(* PLC project KEVIN, Unknown Unnamed 1 *)
(* stored: creationDateTime 2021-12-14T14:39:40, modificationDateTime 2022-01-31T14:09:18 *)

PROGRAM DualCarElevator
  VAR
    C1F1LimitSw AT %IX0.0 : BOOL;
    C2F1LimitSw AT %IX0.1 : BOOL;
    C2F2LimitSw AT %IX0.3 : BOOL;
    C2F3LimitSw AT %IX0.5 : BOOL;
    C2F4LimitSw AT %IX0.7 : BOOL;
    F2DownCall AT %QX0.5 : BOOL;
  END_VAR
  VAR
    C2F1MemLoc : BOOL;
    C2F2MemLoc : BOOL;
    C2F3MemLoc : BOOL;
    C2F4MemLoc : BOOL;
    C2F1VisMem : BOOL;
    C2F2VisMem : BOOL;
    C2F3VisMem : BOOL;
    C2F4VisMem : BOOL;
    C2F1LastVisMem : BOOL;
    C2F2LastVisMem : BOOL;
    C2F3LastVisMem : BOOL;
    C2F4LastVisMem : BOOL;
  END_VAR
  VAR
    C2MotorUp AT %QX0.2 : BOOL;
    C2MotorDown AT %QX0.3 : BOOL;
  END_VAR
  VAR
    C2MotorStops : BOOL;
    C2DoorOpenReady : BOOL;
    C2DoorClose : BOOL;
    C2DoorOpen : BOOL;
    C2DoorIsClosed : BOOL;
    C2DoorCloseReady : BOOL;
  END_VAR
  VAR
    C2F1CarCall AT %QX100.4 : BOOL;
    C2F2CarCall AT %QX100.5 : BOOL;
    C2F3CarCall AT %QX100.6 : BOOL;
    C2F4CarCall AT %QX100.7 : BOOL;
    F2UpCall AT %QX0.6 : BOOL;
    F3UpCall AT %QX1.0 : BOOL;
    F3DownCall AT %QX0.7 : BOOL;
    C1F2LimitSw AT %IX0.2 : BOOL;
    C1F3LimitSw AT %IX0.4 : BOOL;
    C1F4LimitSw AT %IX0.6 : BOOL;
    C1F1CarCall AT %QX100.0 : BOOL;
    C1F2CarCall AT %QX100.1 : BOOL;
    C1F3CarCall AT %QX100.2 : BOOL;
    C1F4CarCall AT %QX100.3 : BOOL;
    F1UpCall AT %QX0.4 : BOOL;
    F4DownCall AT %QX1.1 : BOOL;
    C1MotorUp AT %QX0.0 : BOOL;
    C1MotorDown AT %QX0.1 : BOOL;
  END_VAR
  VAR
    C1MotorStops : BOOL;
    C1DoorOpen : BOOL;
    C1DoorClose : BOOL;
    C1F1MemLoc : BOOL;
    C1F2MemLoc : BOOL;
    C1F3MemLoc : BOOL;
    C1F4MemLoc : BOOL;
    C1F1LastVisMem : BOOL;
    C1F2LastVisMem : BOOL;
    C1F3LastVisMem : BOOL;
    C1F4LastVisMem : BOOL;
    C1F1VisMem : BOOL;
    C1F2VisMem : BOOL;
    C1F3VisMem : BOOL;
    C1F4VisMem : BOOL;
    DoorOpenDelay : TON;
    C1DoorOpenReady : BOOL;
    C1DoorCloseReady : BOOL;
    C1DoorIsClosed : BOOL;
    C1DoorOpeningDelay : TON;
    C1DoorClosingDelay : TON;
    DoorOpenDelay0 : TON;
    C2DoorClosingDelay : TON;
    C2DoorOpeningDelay : TON;
  END_VAR
  VAR
    C1F1CarBtn AT %IX100.0 : BOOL;
    C1F2CarBtn AT %IX100.1 : BOOL;
    C1F3CarBtn AT %IX100.2 : BOOL;
    C1F4CarBtn AT %IX100.3 : BOOL;
    C2F1CarBtn AT %IX100.5 : BOOL;
    C2F2CarBtn AT %IX100.6 : BOOL;
    C2F3CarBtn AT %IX100.7 : BOOL;
    C2F4CarBtn AT %IX101.0 : BOOL;
    F1UpBtn AT %IX1.0 : BOOL;
    F2DownBtn AT %IX1.1 : BOOL;
    F2UpBtn AT %IX1.2 : BOOL;
    F3DownBtn AT %IX1.3 : BOOL;
    F3UpBtn AT %IX1.4 : BOOL;
    F4DownBtn AT %IX1.5 : BOOL;
  END_VAR
  VAR  (* added by the conversion: wires and edge detectors of the diagram *)
    F_TRIG1 : F_TRIG;
    F_TRIG2 : F_TRIG;
    F_TRIG3 : F_TRIG;
    F_TRIG4 : F_TRIG;
    F_TRIG5 : F_TRIG;
    F_TRIG6 : F_TRIG;
    F_TRIG7 : F_TRIG;
    F_TRIG8 : F_TRIG;
  END_VAR

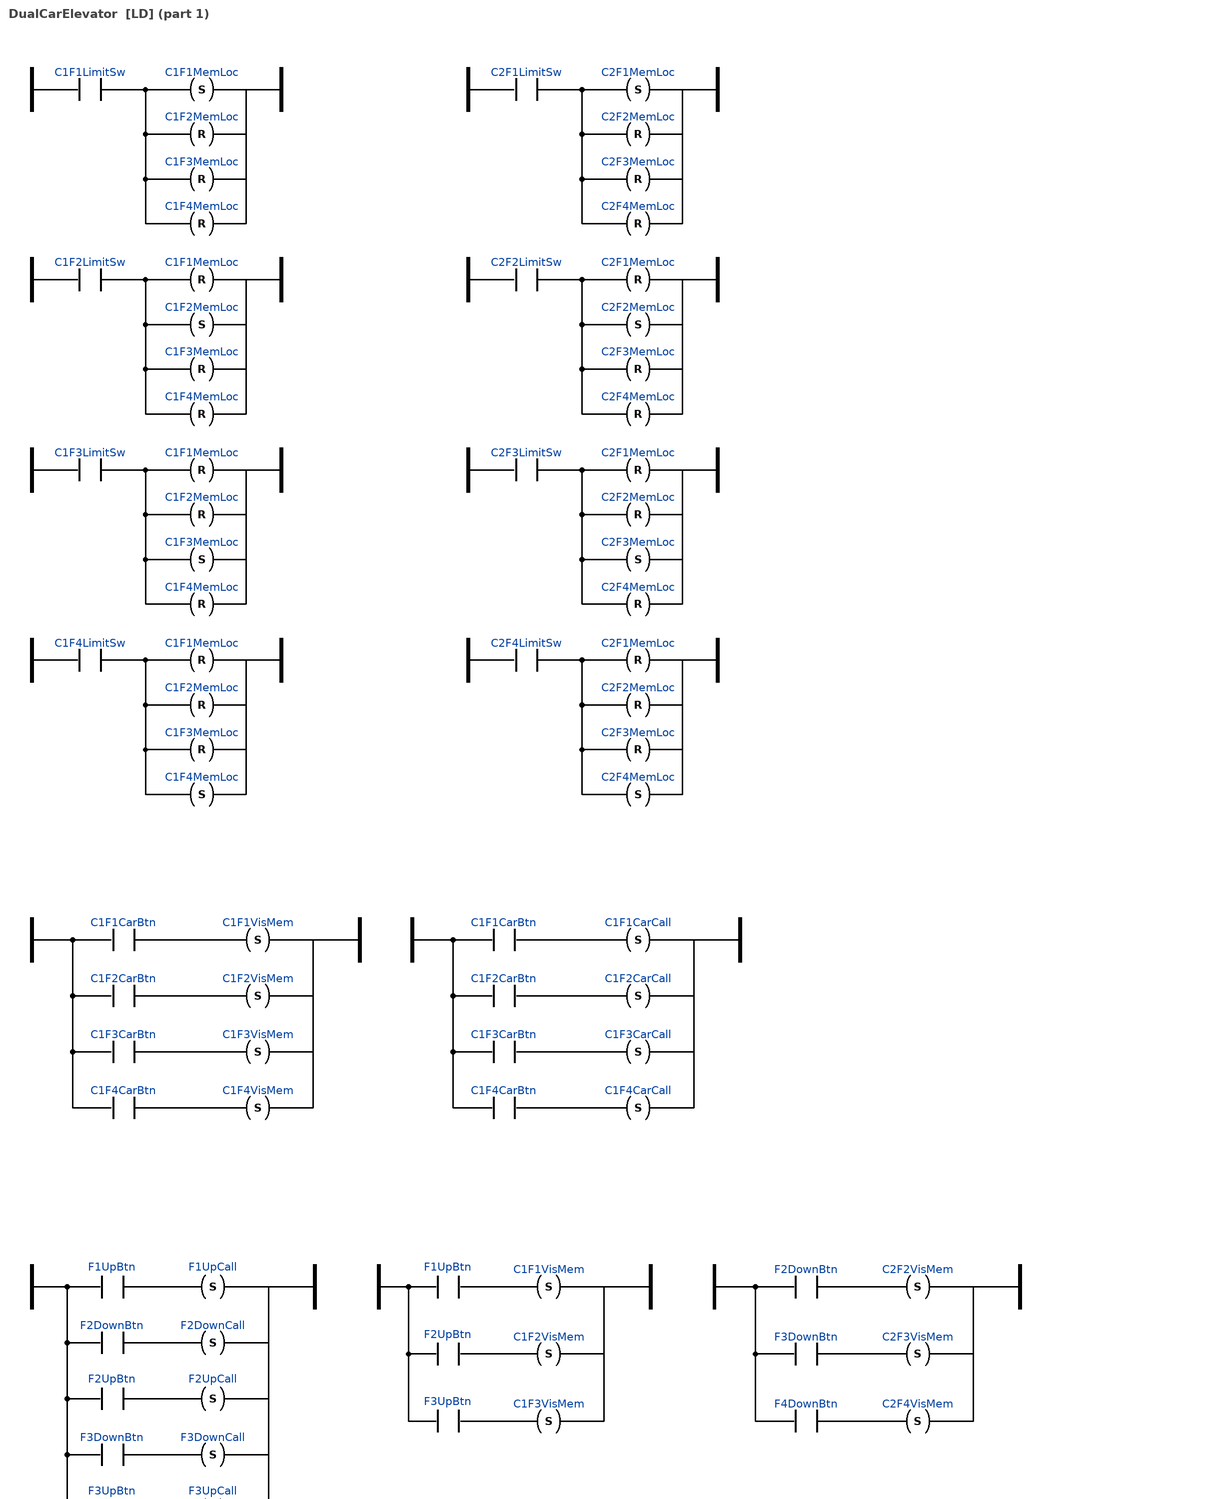
(* LD diagram, written out as Structured Text *)
IF C1F1LimitSw THEN C1F1MemLoc := TRUE; END_IF;
IF C2F1LimitSw THEN C2F1MemLoc := TRUE; END_IF;
IF C1F1LimitSw THEN C1F2MemLoc := FALSE; END_IF;
IF C2F1LimitSw THEN C2F2MemLoc := FALSE; END_IF;
IF C1F1LimitSw THEN C1F3MemLoc := FALSE; END_IF;
IF C2F1LimitSw THEN C2F3MemLoc := FALSE; END_IF;
IF C1F1LimitSw THEN C1F4MemLoc := FALSE; END_IF;
IF C2F1LimitSw THEN C2F4MemLoc := FALSE; END_IF;
IF C1F2LimitSw THEN C1F1MemLoc := FALSE; END_IF;
IF C2F2LimitSw THEN C2F1MemLoc := FALSE; END_IF;
IF C1F2LimitSw THEN C1F2MemLoc := TRUE; END_IF;
IF C2F2LimitSw THEN C2F2MemLoc := TRUE; END_IF;
IF C1F2LimitSw THEN C1F3MemLoc := FALSE; END_IF;
IF C2F2LimitSw THEN C2F3MemLoc := FALSE; END_IF;
IF C1F2LimitSw THEN C1F4MemLoc := FALSE; END_IF;
IF C2F2LimitSw THEN C2F4MemLoc := FALSE; END_IF;
IF C1F3LimitSw THEN C1F1MemLoc := FALSE; END_IF;
IF C2F3LimitSw THEN C2F1MemLoc := FALSE; END_IF;
IF C1F3LimitSw THEN C1F2MemLoc := FALSE; END_IF;
IF C2F3LimitSw THEN C2F2MemLoc := FALSE; END_IF;
IF C1F3LimitSw THEN C1F3MemLoc := TRUE; END_IF;
IF C2F3LimitSw THEN C2F3MemLoc := TRUE; END_IF;
IF C1F3LimitSw THEN C1F4MemLoc := FALSE; END_IF;
IF C2F3LimitSw THEN C2F4MemLoc := FALSE; END_IF;
IF C1F4LimitSw THEN C1F1MemLoc := FALSE; END_IF;
IF C2F4LimitSw THEN C2F1MemLoc := FALSE; END_IF;
IF C1F4LimitSw THEN C1F2MemLoc := FALSE; END_IF;
IF C2F4LimitSw THEN C2F2MemLoc := FALSE; END_IF;
IF C1F4LimitSw THEN C1F3MemLoc := FALSE; END_IF;
IF C2F4LimitSw THEN C2F3MemLoc := FALSE; END_IF;
IF C1F4LimitSw THEN C1F4MemLoc := TRUE; END_IF;
IF C2F4LimitSw THEN C2F4MemLoc := TRUE; END_IF;
IF C1F1CarBtn THEN C1F1VisMem := TRUE; END_IF;
IF C1F1CarBtn THEN C1F1CarCall := TRUE; END_IF;
IF C1F2CarBtn THEN C1F2VisMem := TRUE; END_IF;
IF C1F2CarBtn THEN C1F2CarCall := TRUE; END_IF;
IF C1F3CarBtn THEN C1F3VisMem := TRUE; END_IF;
IF C1F3CarBtn THEN C1F3CarCall := TRUE; END_IF;
IF C1F4CarBtn THEN C1F4VisMem := TRUE; END_IF;
IF C1F4CarBtn THEN C1F4CarCall := TRUE; END_IF;
IF F1UpBtn THEN F1UpCall := TRUE; END_IF;
IF F1UpBtn THEN C1F1VisMem := TRUE; END_IF;
IF F2DownBtn THEN C2F2VisMem := TRUE; END_IF;
IF F2DownBtn THEN F2DownCall := TRUE; END_IF;
IF F2UpBtn THEN C1F2VisMem := TRUE; END_IF;
IF F3DownBtn THEN C2F3VisMem := TRUE; END_IF;
IF F2UpBtn THEN F2UpCall := TRUE; END_IF;
IF F3UpBtn THEN C1F3VisMem := TRUE; END_IF;
IF F4DownBtn THEN C2F4VisMem := TRUE; END_IF;
IF F3DownBtn THEN F3DownCall := TRUE; END_IF;
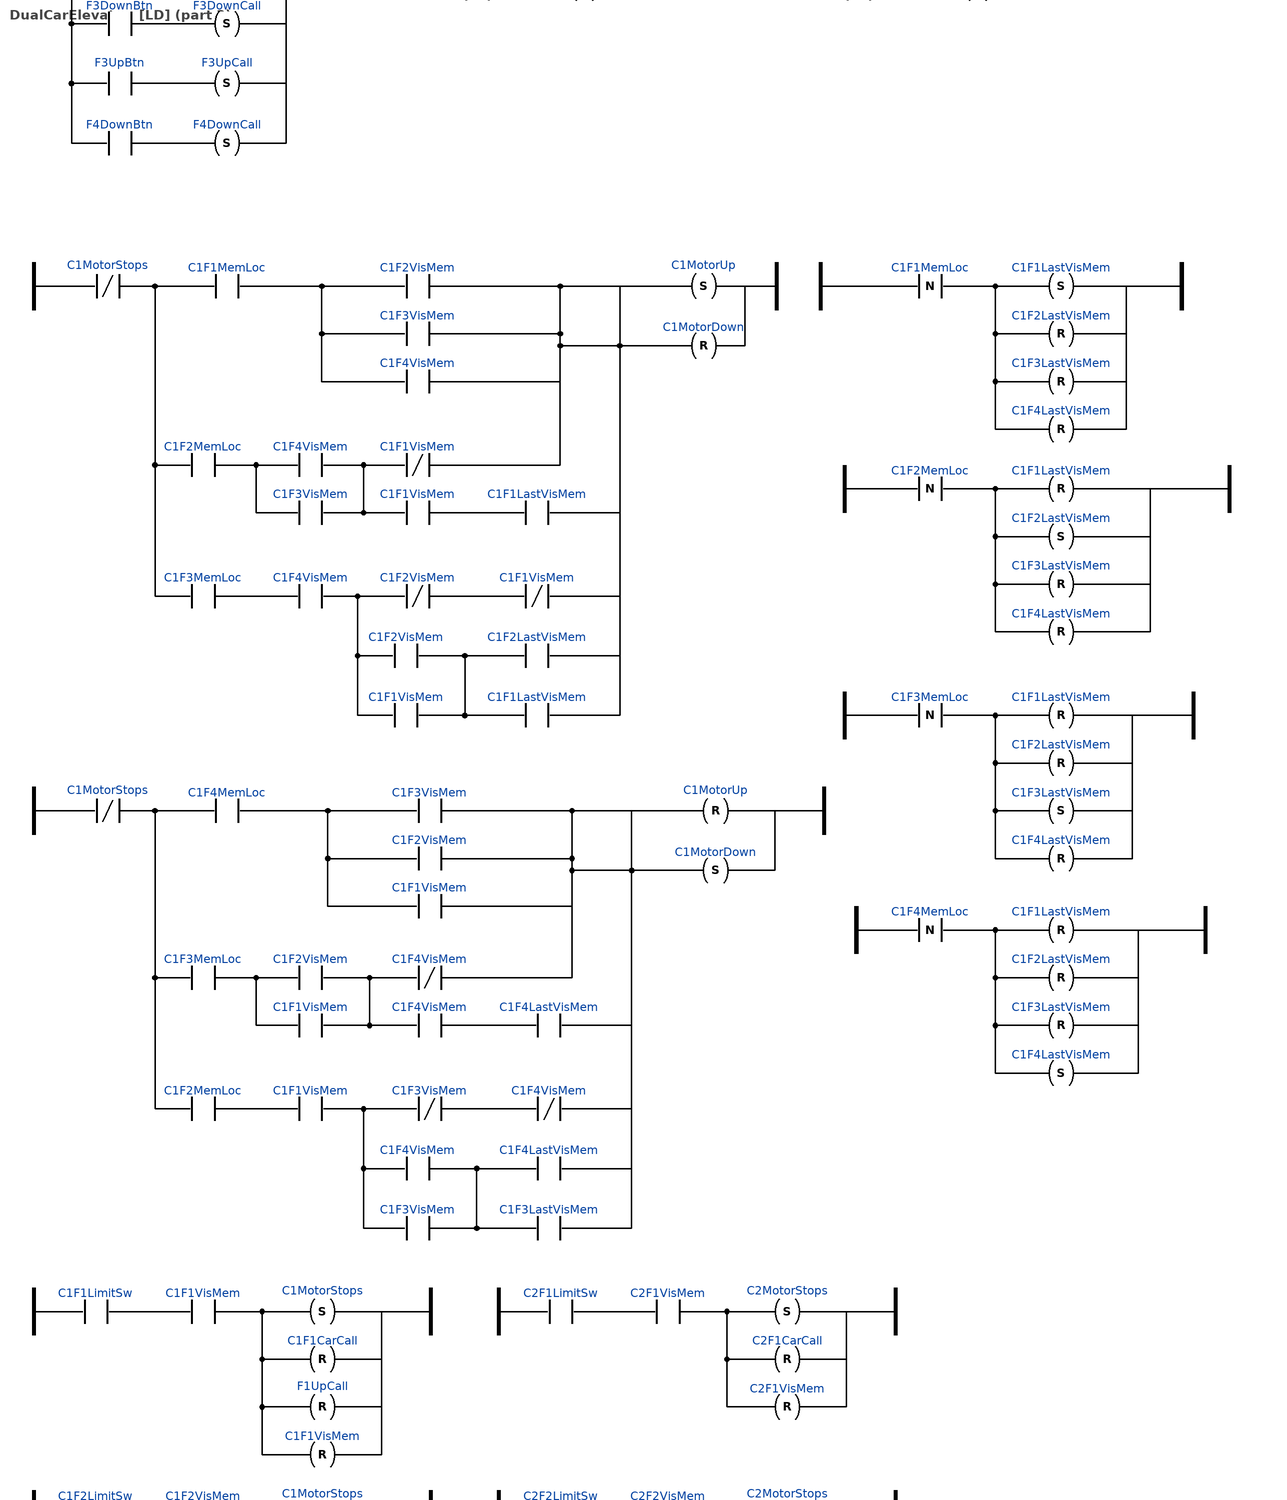
IF F3UpBtn THEN F3UpCall := TRUE; END_IF;
IF F4DownBtn THEN F4DownCall := TRUE; END_IF;
IF NOT C1MotorStops AND (C1F1MemLoc AND C1F2VisMem OR C1F1MemLoc AND C1F3VisMem OR C1F2MemLoc AND (C1F4VisMem OR C1F3VisMem) AND NOT C1F1VisMem OR C1F1MemLoc AND C1F4VisMem OR C1F3MemLoc AND C1F4VisMem AND (C1F2VisMem OR C1F1VisMem) AND C1F2LastVisMem OR C1F2MemLoc AND (C1F4VisMem OR C1F3VisMem) AND C1F1VisMem AND C1F1LastVisMem OR C1F3MemLoc AND C1F4VisMem AND NOT C1F2VisMem AND NOT C1F1VisMem OR C1F3MemLoc AND C1F4VisMem AND (C1F1VisMem OR C1F2VisMem) AND C1F1LastVisMem) THEN C1MotorUp := TRUE; END_IF;
F_TRIG1(CLK := C1F1MemLoc);
IF F_TRIG1.Q THEN C1F1LastVisMem := TRUE; END_IF;
IF F_TRIG1.Q THEN C1F2LastVisMem := FALSE; END_IF;
IF NOT C1MotorStops AND (C1F1MemLoc AND C1F2VisMem OR C1F1MemLoc AND C1F3VisMem OR C1F1MemLoc AND C1F4VisMem OR C1F2MemLoc AND (C1F4VisMem OR C1F3VisMem) AND NOT C1F1VisMem OR C1F2MemLoc AND (C1F4VisMem OR C1F3VisMem) AND C1F1VisMem AND C1F1LastVisMem OR C1F3MemLoc AND C1F4VisMem AND NOT C1F2VisMem AND NOT C1F1VisMem OR C1F3MemLoc AND C1F4VisMem AND (C1F1VisMem OR C1F2VisMem) AND C1F1LastVisMem OR C1F3MemLoc AND C1F4VisMem AND (C1F2VisMem OR C1F1VisMem) AND C1F2LastVisMem) THEN C1MotorDown := FALSE; END_IF;
IF F_TRIG1.Q THEN C1F3LastVisMem := FALSE; END_IF;
IF F_TRIG1.Q THEN C1F4LastVisMem := FALSE; END_IF;
F_TRIG2(CLK := C1F2MemLoc);
IF F_TRIG2.Q THEN C1F1LastVisMem := FALSE; END_IF;
IF F_TRIG2.Q THEN C1F2LastVisMem := TRUE; END_IF;
IF F_TRIG2.Q THEN C1F3LastVisMem := FALSE; END_IF;
IF F_TRIG2.Q THEN C1F4LastVisMem := FALSE; END_IF;
F_TRIG3(CLK := C1F3MemLoc);
IF F_TRIG3.Q THEN C1F1LastVisMem := FALSE; END_IF;
IF F_TRIG3.Q THEN C1F2LastVisMem := FALSE; END_IF;
IF NOT C1MotorStops AND (C1F4MemLoc AND C1F3VisMem OR C1F4MemLoc AND C1F2VisMem OR C1F4MemLoc AND C1F1VisMem OR C1F3MemLoc AND (C1F1VisMem OR C1F2VisMem) AND NOT C1F4VisMem OR C1F3MemLoc AND (C1F1VisMem OR C1F2VisMem) AND C1F4VisMem AND C1F4LastVisMem OR C1F2MemLoc AND C1F1VisMem AND NOT C1F3VisMem AND NOT C1F4VisMem OR C1F2MemLoc AND C1F1VisMem AND (C1F4VisMem OR C1F3VisMem) AND C1F4LastVisMem OR C1F2MemLoc AND C1F1VisMem AND (C1F3VisMem OR C1F4VisMem) AND C1F3LastVisMem) THEN C1MotorUp := FALSE; END_IF;
IF F_TRIG3.Q THEN C1F3LastVisMem := TRUE; END_IF;
IF F_TRIG3.Q THEN C1F4LastVisMem := FALSE; END_IF;
IF NOT C1MotorStops AND (C1F4MemLoc AND C1F3VisMem OR C1F4MemLoc AND C1F2VisMem OR C1F4MemLoc AND C1F1VisMem OR C1F3MemLoc AND (C1F1VisMem OR C1F2VisMem) AND NOT C1F4VisMem OR C1F3MemLoc AND (C1F1VisMem OR C1F2VisMem) AND C1F4VisMem AND C1F4LastVisMem OR C1F2MemLoc AND C1F1VisMem AND NOT C1F3VisMem AND NOT C1F4VisMem OR C1F2MemLoc AND C1F1VisMem AND (C1F3VisMem OR C1F4VisMem) AND C1F3LastVisMem OR C1F2MemLoc AND C1F1VisMem AND (C1F4VisMem OR C1F3VisMem) AND C1F4LastVisMem) THEN C1MotorDown := TRUE; END_IF;
F_TRIG4(CLK := C1F4MemLoc);
IF F_TRIG4.Q THEN C1F1LastVisMem := FALSE; END_IF;
IF F_TRIG4.Q THEN C1F2LastVisMem := FALSE; END_IF;
IF F_TRIG4.Q THEN C1F3LastVisMem := FALSE; END_IF;
IF F_TRIG4.Q THEN C1F4LastVisMem := TRUE; END_IF;
IF C1F1LimitSw AND C1F1VisMem THEN C1MotorStops := TRUE; END_IF;
IF C2F1LimitSw AND C2F1VisMem THEN C2MotorStops := TRUE; END_IF;
IF C1F1LimitSw AND C1F1VisMem THEN C1F1CarCall := FALSE; END_IF;
IF C2F1LimitSw AND C2F1VisMem THEN C2F1CarCall := FALSE; END_IF;
IF C1F1LimitSw AND C1F1VisMem THEN F1UpCall := FALSE; END_IF;
IF C2F1LimitSw AND C2F1VisMem THEN C2F1VisMem := FALSE; END_IF;
IF C1F1LimitSw AND C1F1VisMem THEN C1F1VisMem := FALSE; END_IF;
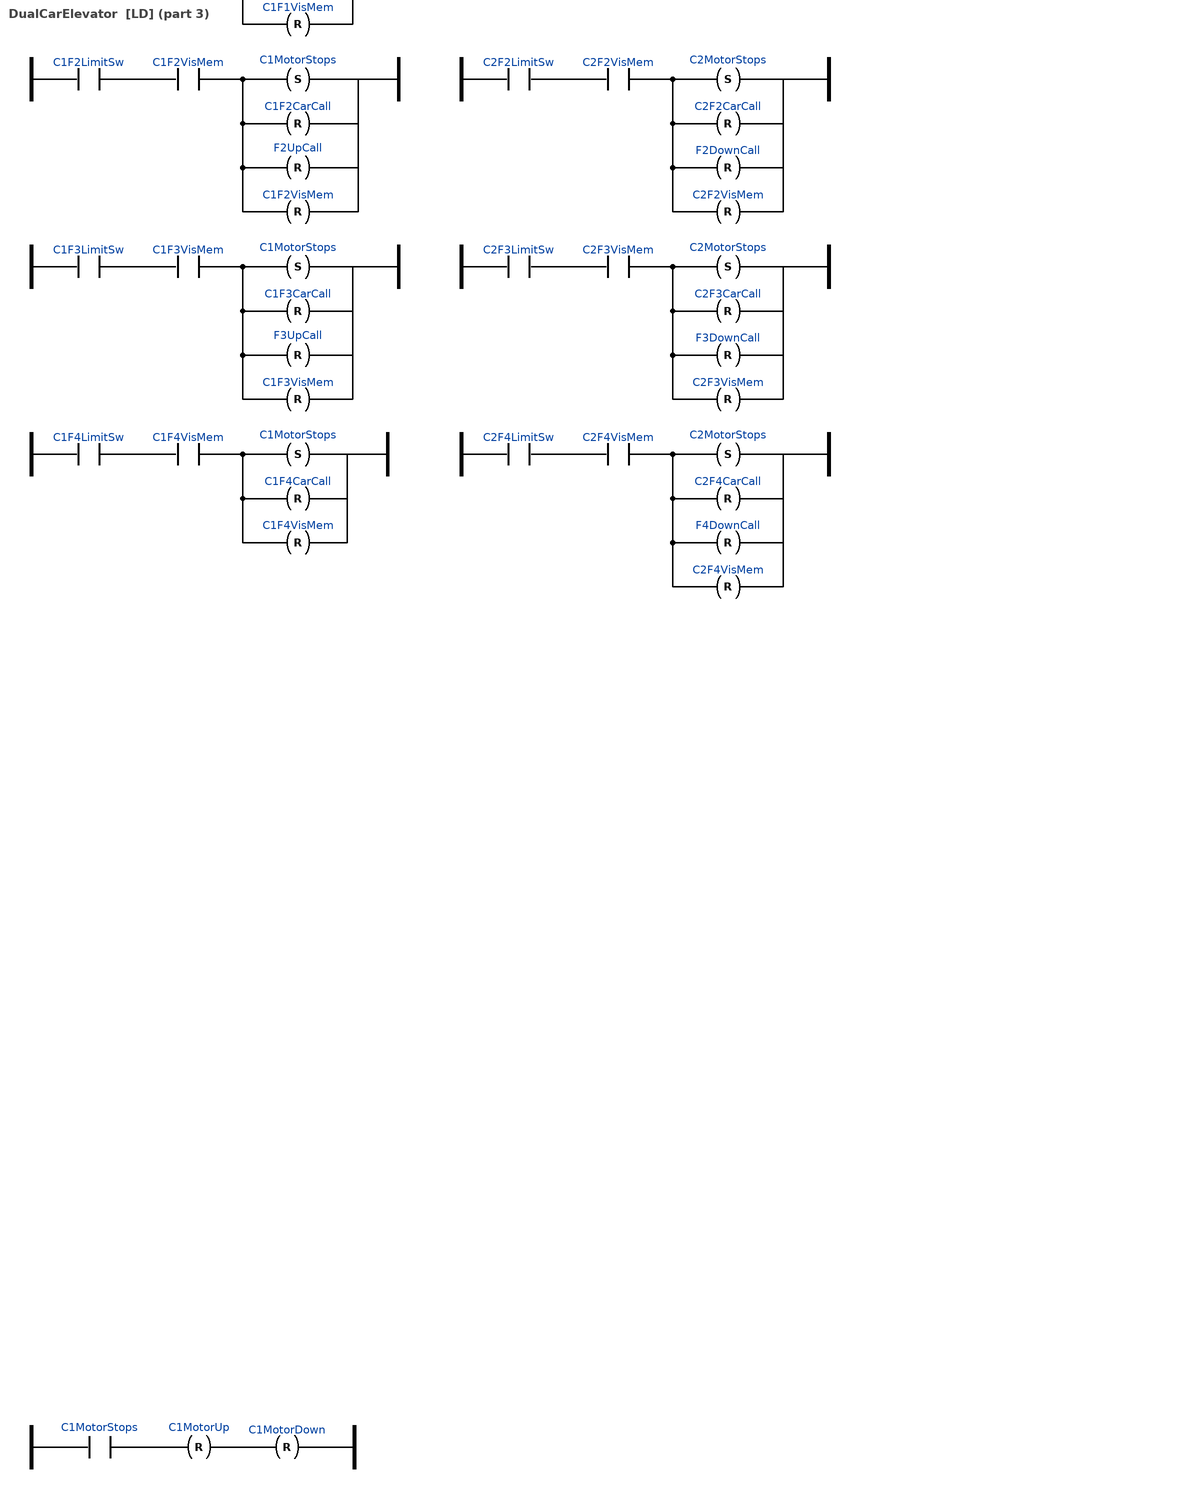
IF C1F2LimitSw AND C1F2VisMem THEN C1MotorStops := TRUE; END_IF;
IF C2F2LimitSw AND C2F2VisMem THEN C2MotorStops := TRUE; END_IF;
IF C1F2LimitSw AND C1F2VisMem THEN C1F2CarCall := FALSE; END_IF;
IF C2F2LimitSw AND C2F2VisMem THEN C2F2CarCall := FALSE; END_IF;
IF C1F2LimitSw AND C1F2VisMem THEN F2UpCall := FALSE; END_IF;
IF C2F2LimitSw AND C2F2VisMem THEN F2DownCall := FALSE; END_IF;
IF C1F2LimitSw AND C1F2VisMem THEN C1F2VisMem := FALSE; END_IF;
IF C2F2LimitSw AND C2F2VisMem THEN C2F2VisMem := FALSE; END_IF;
IF C1F3LimitSw AND C1F3VisMem THEN C1MotorStops := TRUE; END_IF;
IF C2F3LimitSw AND C2F3VisMem THEN C2MotorStops := TRUE; END_IF;
IF C1F3LimitSw AND C1F3VisMem THEN C1F3CarCall := FALSE; END_IF;
IF C2F3LimitSw AND C2F3VisMem THEN C2F3CarCall := FALSE; END_IF;
IF C1F3LimitSw AND C1F3VisMem THEN F3UpCall := FALSE; END_IF;
IF C2F3LimitSw AND C2F3VisMem THEN F3DownCall := FALSE; END_IF;
IF C1F3LimitSw AND C1F3VisMem THEN C1F3VisMem := FALSE; END_IF;
IF C2F3LimitSw AND C2F3VisMem THEN C2F3VisMem := FALSE; END_IF;
IF C1F4LimitSw AND C1F4VisMem THEN C1MotorStops := TRUE; END_IF;
IF C2F4LimitSw AND C2F4VisMem THEN C2MotorStops := TRUE; END_IF;
IF C1F4LimitSw AND C1F4VisMem THEN C1F4CarCall := FALSE; END_IF;
IF C2F4LimitSw AND C2F4VisMem THEN C2F4CarCall := FALSE; END_IF;
IF C1F4LimitSw AND C1F4VisMem THEN C1F4VisMem := FALSE; END_IF;
IF C2F4LimitSw AND C2F4VisMem THEN F4DownCall := FALSE; END_IF;
IF C2F4LimitSw AND C2F4VisMem THEN C2F4VisMem := FALSE; END_IF;
IF C1MotorStops THEN C1MotorUp := FALSE; END_IF;
IF C1MotorStops THEN C1MotorDown := FALSE; END_IF;
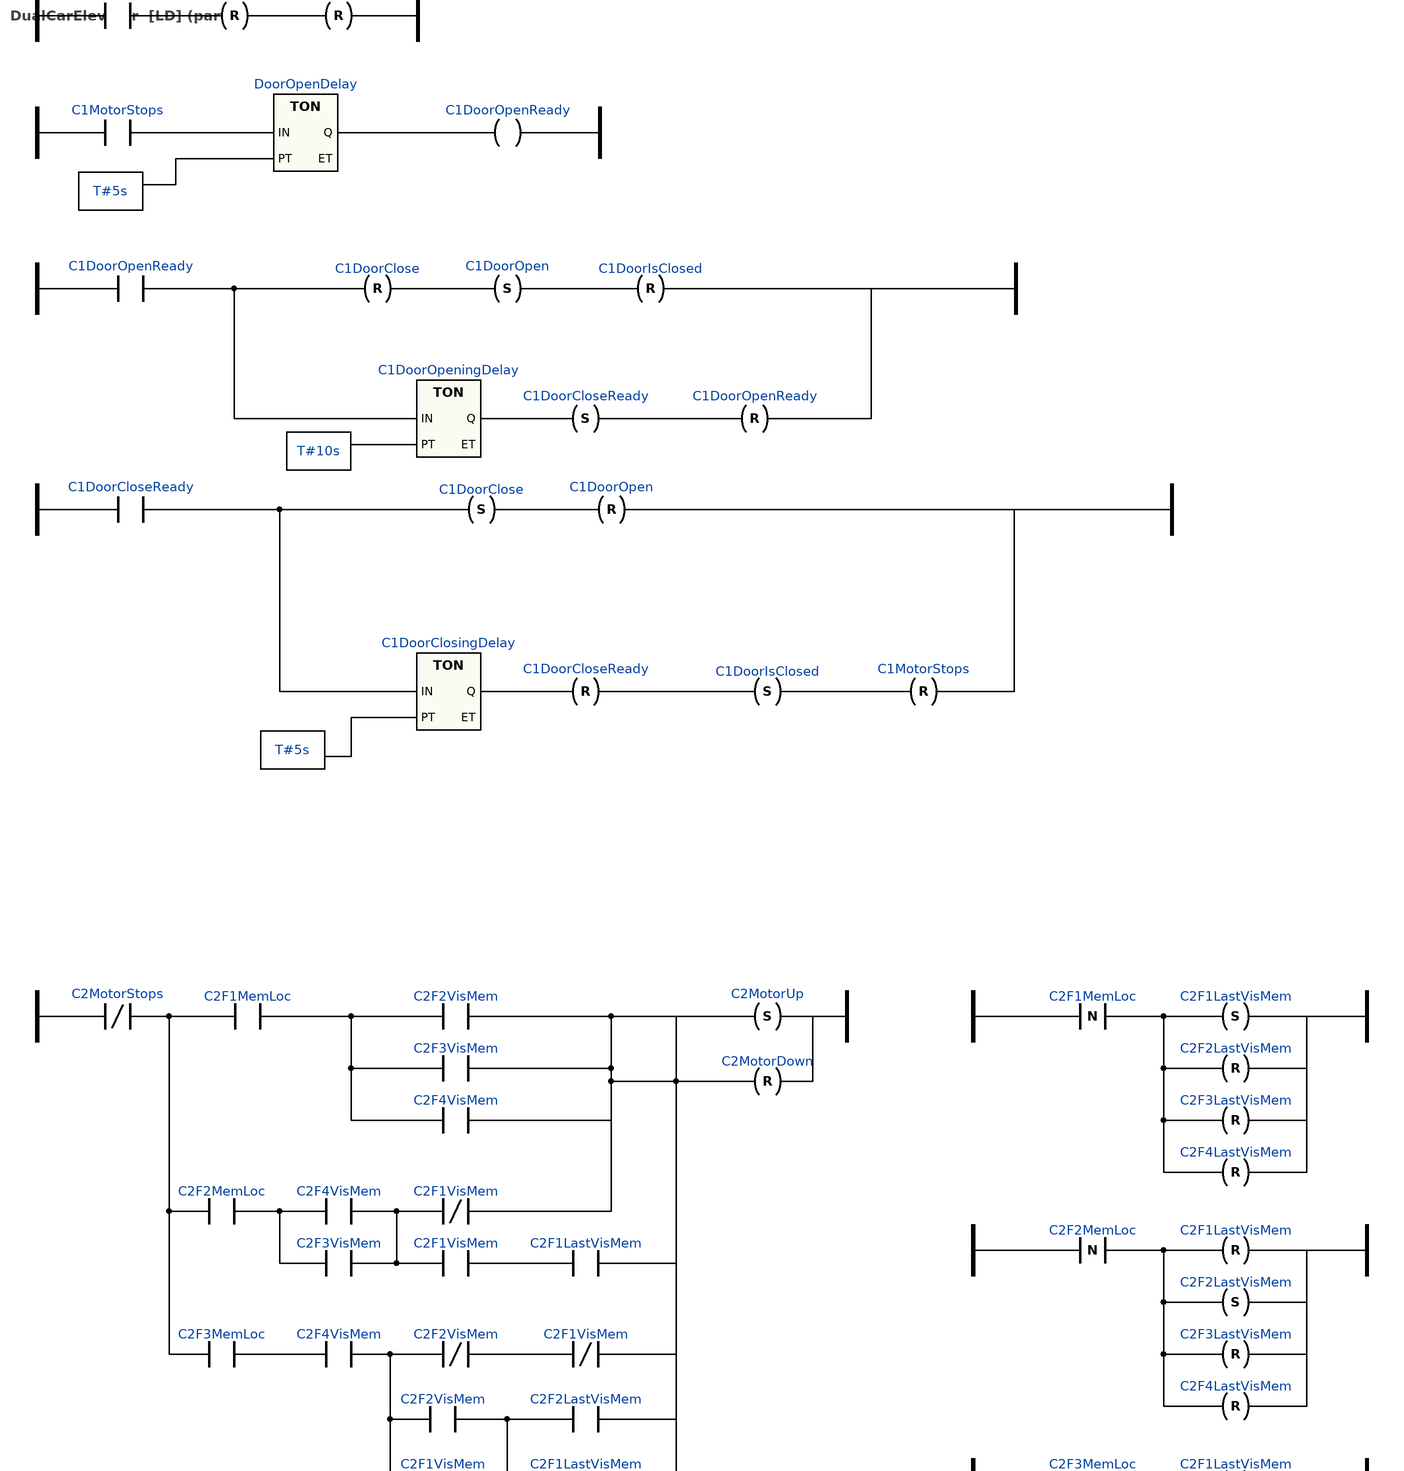
DoorOpenDelay(IN := C1MotorStops, PT := T#5s);
C1DoorOpenReady := DoorOpenDelay.Q;
IF C1DoorOpenReady THEN C1DoorClose := FALSE; END_IF;
IF C1DoorOpenReady THEN C1DoorOpen := TRUE; END_IF;
IF C1DoorOpenReady THEN C1DoorIsClosed := FALSE; END_IF;
C1DoorOpeningDelay(IN := C1DoorOpenReady, PT := T#10s);
IF C1DoorOpeningDelay.Q THEN C1DoorCloseReady := TRUE; END_IF;
IF C1DoorOpeningDelay.Q THEN C1DoorOpenReady := FALSE; END_IF;
IF C1DoorCloseReady THEN C1DoorClose := TRUE; END_IF;
IF C1DoorCloseReady THEN C1DoorOpen := FALSE; END_IF;
C1DoorClosingDelay(IN := C1DoorCloseReady, PT := T#5s);
IF C1DoorClosingDelay.Q THEN C1DoorCloseReady := FALSE; END_IF;
IF C1DoorClosingDelay.Q THEN C1DoorIsClosed := TRUE; END_IF;
IF C1DoorClosingDelay.Q THEN C1MotorStops := FALSE; END_IF;
IF NOT C2MotorStops AND (C2F1MemLoc AND C2F2VisMem OR C2F1MemLoc AND C2F3VisMem OR C2F2MemLoc AND (C2F4VisMem OR C2F3VisMem) AND NOT C2F1VisMem OR C2F1MemLoc AND C2F4VisMem OR C2F3MemLoc AND C2F4VisMem AND (C2F2VisMem OR C2F1VisMem) AND C2F2LastVisMem OR C2F2MemLoc AND (C2F4VisMem OR C2F3VisMem) AND C2F1VisMem AND C2F1LastVisMem OR C2F3MemLoc AND C2F4VisMem AND NOT C2F2VisMem AND NOT C2F1VisMem OR C2F3MemLoc AND C2F4VisMem AND (C2F1VisMem OR C2F2VisMem) AND C2F1LastVisMem) THEN C2MotorUp := TRUE; END_IF;
F_TRIG5(CLK := C2F1MemLoc);
IF F_TRIG5.Q THEN C2F1LastVisMem := TRUE; END_IF;
IF F_TRIG5.Q THEN C2F2LastVisMem := FALSE; END_IF;
IF NOT C2MotorStops AND (C2F1MemLoc AND C2F2VisMem OR C2F1MemLoc AND C2F3VisMem OR C2F1MemLoc AND C2F4VisMem OR C2F2MemLoc AND (C2F4VisMem OR C2F3VisMem) AND NOT C2F1VisMem OR C2F2MemLoc AND (C2F4VisMem OR C2F3VisMem) AND C2F1VisMem AND C2F1LastVisMem OR C2F3MemLoc AND C2F4VisMem AND NOT C2F2VisMem AND NOT C2F1VisMem OR C2F3MemLoc AND C2F4VisMem AND (C2F2VisMem OR C2F1VisMem) AND C2F2LastVisMem OR C2F3MemLoc AND C2F4VisMem AND (C2F1VisMem OR C2F2VisMem) AND C2F1LastVisMem) THEN C2MotorDown := FALSE; END_IF;
IF F_TRIG5.Q THEN C2F3LastVisMem := FALSE; END_IF;
IF F_TRIG5.Q THEN C2F4LastVisMem := FALSE; END_IF;
F_TRIG6(CLK := C2F2MemLoc);
IF F_TRIG6.Q THEN C2F1LastVisMem := FALSE; END_IF;
IF F_TRIG6.Q THEN C2F2LastVisMem := TRUE; END_IF;
IF F_TRIG6.Q THEN C2F3LastVisMem := FALSE; END_IF;
IF F_TRIG6.Q THEN C2F4LastVisMem := FALSE; END_IF;
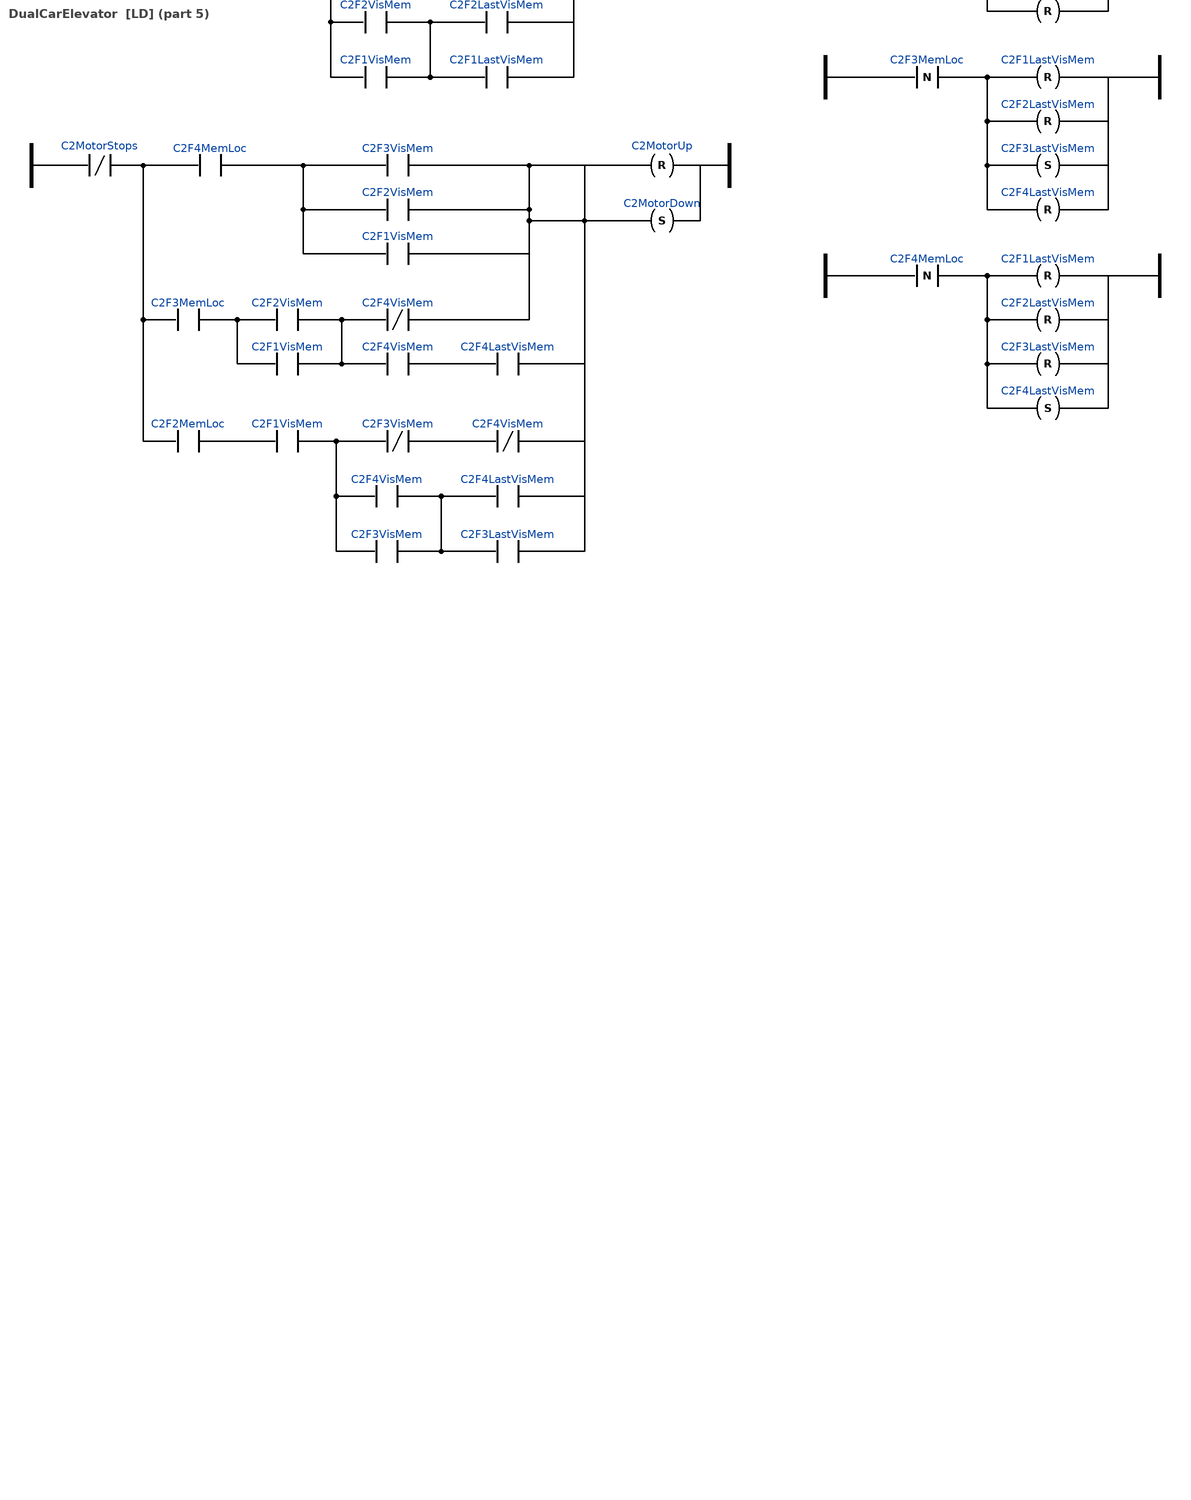
F_TRIG7(CLK := C2F3MemLoc);
IF F_TRIG7.Q THEN C2F1LastVisMem := FALSE; END_IF;
IF F_TRIG7.Q THEN C2F2LastVisMem := FALSE; END_IF;
IF NOT C2MotorStops AND (C2F4MemLoc AND C2F3VisMem OR C2F4MemLoc AND C2F1VisMem OR C2F3MemLoc AND (C2F1VisMem OR C2F2VisMem) AND NOT C2F4VisMem OR C2F4MemLoc AND C2F2VisMem OR C2F3MemLoc AND (C2F1VisMem OR C2F2VisMem) AND C2F4VisMem AND C2F4LastVisMem OR C2F2MemLoc AND C2F1VisMem AND NOT C2F3VisMem AND NOT C2F4VisMem OR C2F2MemLoc AND C2F1VisMem AND (C2F3VisMem OR C2F4VisMem) AND C2F3LastVisMem OR C2F2MemLoc AND C2F1VisMem AND (C2F4VisMem OR C2F3VisMem) AND C2F4LastVisMem) THEN C2MotorUp := FALSE; END_IF;
IF F_TRIG7.Q THEN C2F3LastVisMem := TRUE; END_IF;
IF F_TRIG7.Q THEN C2F4LastVisMem := FALSE; END_IF;
IF NOT C2MotorStops AND (C2F4MemLoc AND C2F3VisMem OR C2F4MemLoc AND C2F2VisMem OR C2F4MemLoc AND C2F1VisMem OR C2F3MemLoc AND (C2F1VisMem OR C2F2VisMem) AND NOT C2F4VisMem OR C2F3MemLoc AND (C2F1VisMem OR C2F2VisMem) AND C2F4VisMem AND C2F4LastVisMem OR C2F2MemLoc AND C2F1VisMem AND NOT C2F3VisMem AND NOT C2F4VisMem OR C2F2MemLoc AND C2F1VisMem AND (C2F3VisMem OR C2F4VisMem) AND C2F3LastVisMem OR C2F2MemLoc AND C2F1VisMem AND (C2F4VisMem OR C2F3VisMem) AND C2F4LastVisMem) THEN C2MotorDown := TRUE; END_IF;
F_TRIG8(CLK := C2F4MemLoc);
IF F_TRIG8.Q THEN C2F1LastVisMem := FALSE; END_IF;
IF F_TRIG8.Q THEN C2F2LastVisMem := FALSE; END_IF;
IF F_TRIG8.Q THEN C2F3LastVisMem := FALSE; END_IF;
IF F_TRIG8.Q THEN C2F4LastVisMem := TRUE; END_IF;
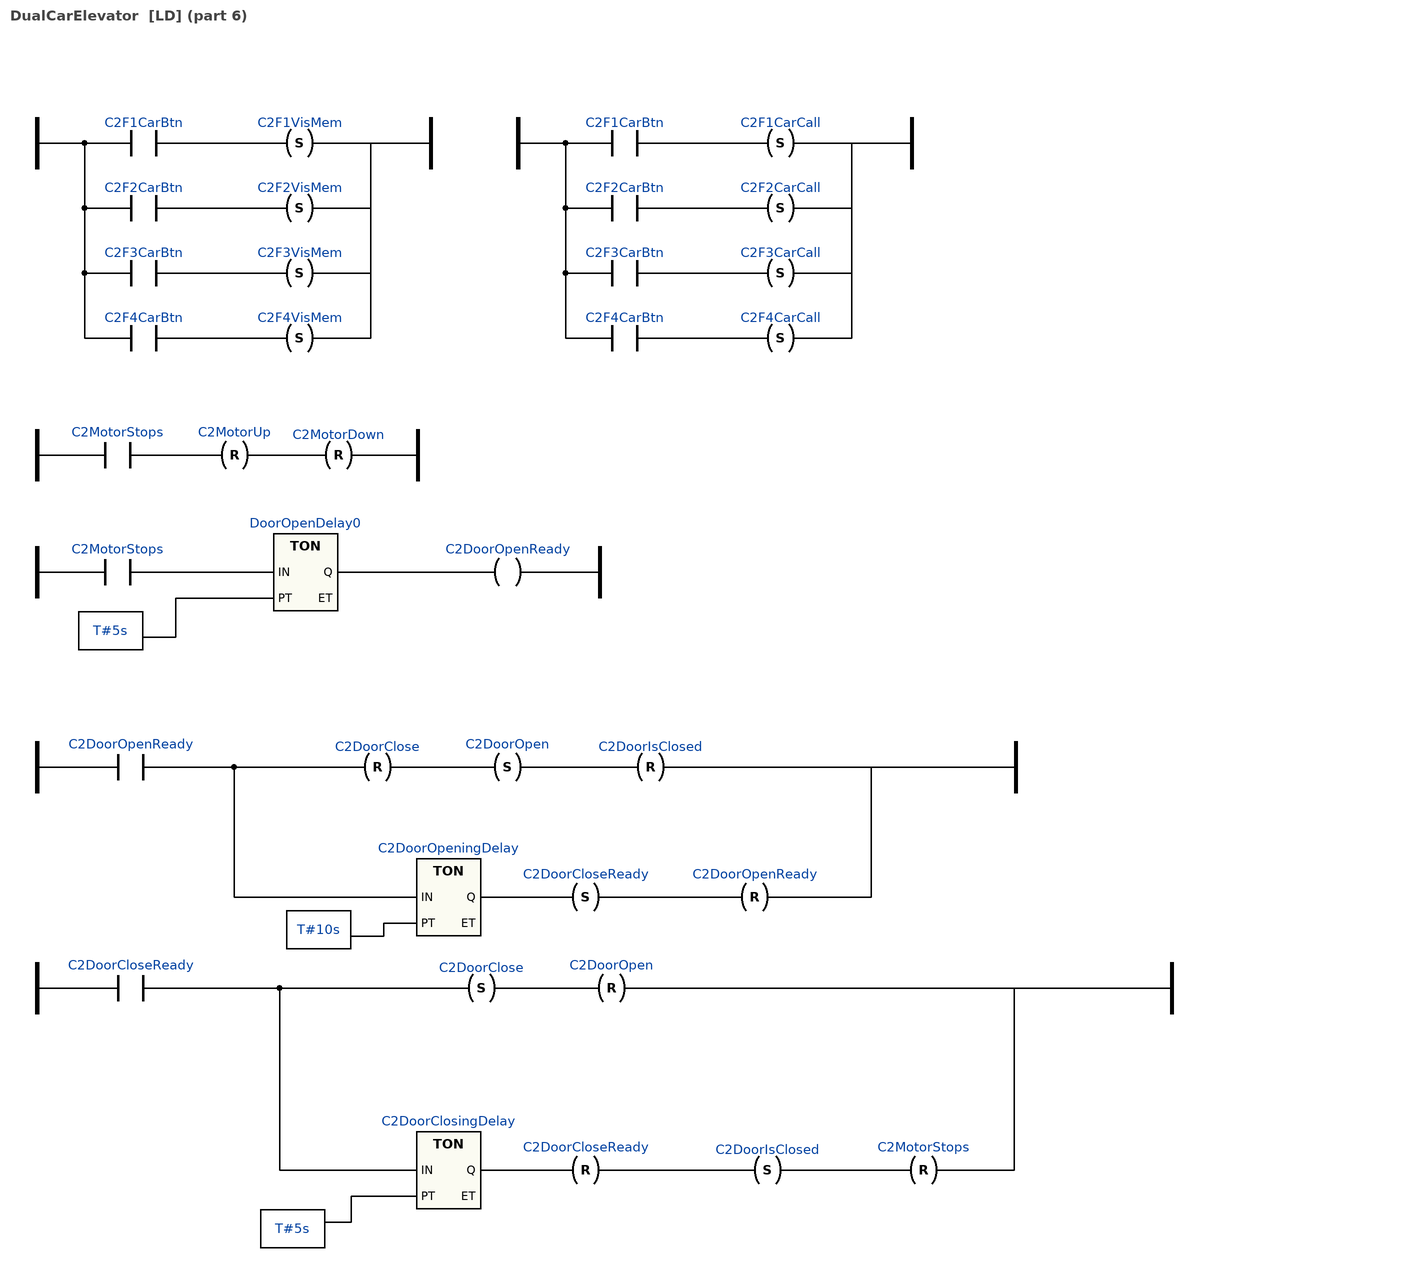
IF C2F1CarBtn THEN C2F1VisMem := TRUE; END_IF;
IF C2F1CarBtn THEN C2F1CarCall := TRUE; END_IF;
IF C2F2CarBtn THEN C2F2VisMem := TRUE; END_IF;
IF C2F2CarBtn THEN C2F2CarCall := TRUE; END_IF;
IF C2F3CarBtn THEN C2F3VisMem := TRUE; END_IF;
IF C2F3CarBtn THEN C2F3CarCall := TRUE; END_IF;
IF C2F4CarBtn THEN C2F4VisMem := TRUE; END_IF;
IF C2F4CarBtn THEN C2F4CarCall := TRUE; END_IF;
IF C2MotorStops THEN C2MotorUp := FALSE; END_IF;
IF C2MotorStops THEN C2MotorDown := FALSE; END_IF;
DoorOpenDelay0(IN := C2MotorStops, PT := T#5s);
C2DoorOpenReady := DoorOpenDelay0.Q;
IF C2DoorOpenReady THEN C2DoorClose := FALSE; END_IF;
IF C2DoorOpenReady THEN C2DoorOpen := TRUE; END_IF;
IF C2DoorOpenReady THEN C2DoorIsClosed := FALSE; END_IF;
C2DoorOpeningDelay(IN := C2DoorOpenReady, PT := T#10s);
IF C2DoorOpeningDelay.Q THEN C2DoorCloseReady := TRUE; END_IF;
IF C2DoorOpeningDelay.Q THEN C2DoorOpenReady := FALSE; END_IF;
IF C2DoorCloseReady THEN C2DoorClose := TRUE; END_IF;
IF C2DoorCloseReady THEN C2DoorOpen := FALSE; END_IF;
C2DoorClosingDelay(IN := C2DoorCloseReady, PT := T#5s);
IF C2DoorClosingDelay.Q THEN C2DoorCloseReady := FALSE; END_IF;
IF C2DoorClosingDelay.Q THEN C2DoorIsClosed := TRUE; END_IF;
IF C2DoorClosingDelay.Q THEN C2MotorStops := FALSE; END_IF;
END_PROGRAM

CONFIGURATION Config0
  RESOURCE Res0 ON PLC
    TASK task0(INTERVAL := T#20ms, PRIORITY := 0);
    PROGRAM instance0 WITH task0 : DualCarElevator;
  END_RESOURCE
END_CONFIGURATION
